FUNCTION Convert_ULINT_TO_SINT : Hresult
VAR_INPUT
	in : ULINT;
	out : REFERENCE TO SINT;
END_VAR
VAR
	converted : SINT;
END_VAR
VAR CONSTANT
	INCOMPATIBLE : HRESULT := 16#9811070E;
END_VAR

converted := ULINT_TO_SINT(in);

IF (SINT_TO_ULINT(converted) <> in) THEN
	Convert_ULINT_TO_SINT := INCOMPATIBLE;
	RETURN;
END_IF

out := converted;

END_FUNCTION

(* stored: Version 1.1.0.1, ProductVersion 3.1.4024.12
   POU Convert_ULINT_TO_SINT: Id {200cf821-9203-4afd-9ce5-b288572f78a3}, SpecialFunc None *)
